# EPICS substitutions: epics/m-epics-eemcu/eemcuApp/Db/Sim8-extra-m7.substitutions
file "eemcu-extra.template"
{
pattern
{P,      M,    R,   PORT, ADDR, PREC, HOMEPROC}
{IOC:,   m7, m7-,   MCU1,    7, 3,    3}
}
